// TIA Portal V18 export
VAR_GLOBAL   // PLC tag table "RemoteIO_DI_1"
   "iA-Loading-02Detection" AT %I1000.0 : Bool;   // A-转盘上料-02切料位检测
   "iA-Loading-02GripperTakeDetection" AT %I1000.1 : Bool;   // A-转盘上料-02夹爪取料位检测
   "iA-Loading-02PipeDetection" AT %I1000.2 : Bool;   // A-转盘上料-02料管检测
   "RESERVE_I1000.3" AT %I1000.3 : Bool;   // 备用_I1000.3
   "iA-Loading-02HorizontalCylinderInWP" AT %I1000.4 : Bool;   // A-转盘上料-02水平移栽气缸工作位
   "iA-Loading-02HorizontalCylinderInHP" AT %I1000.5 : Bool;   // A-转盘上料-02水平移栽气缸原始位
   "iA-Loading-02UpDownTakeCylinderInWP" AT %I1000.6 : Bool;   // A-转盘上料-02上下取料气缸工作位
   "iA-Loading-02UpDownTakeCylinderInHP" AT %I1000.7 : Bool;   // A-转盘上料-02上下取料气缸原始位
   "iB-PressFitting-02GripperCylinderInWP" AT %I1001.0 : Bool;   // B-压装模组-02夹爪气缸工作位
   "iB-PressFitting-02GripperCylinderInHP" AT %I1001.1 : Bool;   // B-压装模组-02夹爪气缸原始位
   "iB-PressFitting-02DownRingDetection" AT %I1001.2 : Bool;   // 备用_I1001.2
   "RESERVE_I1001.3" AT %I1001.3 : Bool;   // 备用_I1001.3
   "RESERVE_I1001.4" AT %I1001.4 : Bool;   // 备用_I1001.4
   "RESERVE_I1001.5" AT %I1001.5 : Bool;   // 备用_I1001.5
   "RESERVE_I1001.6" AT %I1001.6 : Bool;   // 备用_I1001.6
   "RESERVE_I1001.7" AT %I1001.7 : Bool;   // 备用_I1001.7
   "iB-PressFitting-02CylinderInWP" AT %I1002.0 : Bool;   // B-压装模组-02中转气缸工作位
   "iB-PressFitting-02CylinderInHP" AT %I1002.1 : Bool;   // B-压装模组-02中转气缸原始位
   "iB-PressFitting-02UpRingDetection" AT %I1002.2 : Bool;   // B-压装模组-02shaft有无检测
   "iB-PressFitting-02ShaftDetection" AT %I1002.3 : Bool;   // B-压装模组-02ring有无检测
   "RESERVE_I1002.4" AT %I1002.4 : Bool;   // 备用_I1002.4
   "RESERVE_I1002.5" AT %I1002.5 : Bool;   // 备用_I1002.5
   "RESERVE_I1002.6" AT %I1002.6 : Bool;   // 备用_I1002.6
   "RESERVE_I1002.7" AT %I1002.7 : Bool;   // 备用_I1002.7
   "iE-NG-02NGLocationCylinderInWP" AT %I1003.0 : Bool;   // E-NG料盒-02NG定位气缸工作位
   "iE-NG-02NGLocationCylinderInHP" AT %I1003.1 : Bool;   // E-NG料盒-02NG定位气缸原始位
   "iE-NG-03ShaftDispenseNGDetection" AT %I1003.2 : Bool;   // E-NG中转位-03shaft点胶NG有无检测
   "iE-NG-03MagnetDispenseNGDetection" AT %I1003.3 : Bool;   // E-NG中转位-03magnet点胶NG有无检测
   "iE-NG-02Detection" AT %I1003.4 : Bool;   // E-NG料盒-02到位检测
   "iC-GlueServoHomePos" AT %I1003.5 : Bool;   // 备用_I1003.5 / C-涂胶伺服原点
   "RESERVE_I1003.6" AT %I1003.6 : Bool;   // 备用_I1003.6
   "RESERVE_I1003.7" AT %I1003.7 : Bool;   // 备用_I1003.7
   "iC-LocationCylinderInWP" AT %I1004.0 : Bool;   // C-涂胶定位模组标准气缸工作位
   "iC-LocationCylinderInHP" AT %I1004.1 : Bool;   // C-涂胶定位模组标准气缸原始位
   "iC-LocationShaftDetection" AT %I1004.2 : Bool;   // C-涂胶定位模组shaft有无检测
   "iE-NG-01Detection" AT %I1004.3 : Bool;   // 备用_I1004.3 / E-NG料盒-01到位检测
   "iE-NG-01NGLocationCylinderInWP" AT %I1004.4 : Bool;   // E-NG料盒-01NG定位气缸工作位
   "iE-NG-01NGLocationCylinderInHP" AT %I1004.5 : Bool;   // E-NG料盒-01NG定位气缸原始位
   "RESERVE_I1004.6" AT %I1004.6 : Bool;   // E-NG料盒-01到位检测 / 备用_I1004.6
   "RESERVE_I1004.7" AT %I1004.7 : Bool;   // 备用_I1004.7
   "iB-PressFitting-01GripperCylinderInWP" AT %I1005.0 : Bool;   // B-压装模组-01夹爪气缸工作位
   "iB-PressFitting-01GripperCylinderInHP" AT %I1005.1 : Bool;   // B-压装模组-01夹爪气缸原始位
   "iB-PressFitting-01DownRingDetection" AT %I1005.2 : Bool;   // 备用_I1005.2
   "RESERVE_I1005.3" AT %I1005.3 : Bool;   // 备用_I1005.3
   "RESERVE_I1005.4" AT %I1005.4 : Bool;   // 备用_I1005.4
   "RESERVE_I1005.5" AT %I1005.5 : Bool;   // 备用_I1005.5
   "RESERVE_I1005.6" AT %I1005.6 : Bool;   // 备用_I1005.6
   "RESERVE_I1005.7" AT %I1005.7 : Bool;   // 备用_I1005.7
   "iB-PressFitting-01CylinderInWP" AT %I1006.0 : Bool;   // B-压装模组-01中转气缸工作位
   "iB-PressFitting-01CylinderInHP" AT %I1006.1 : Bool;   // B-压装模组-01中转气缸原始位
   "iB-PressFitting-01UpRingDetection" AT %I1006.2 : Bool;   // B-压装模组-01shaft有无检测-05
   "iB-PressFitting-01ShaftDetection" AT %I1006.3 : Bool;   // B-压装模组-01ring有无检测-06
   "iA-Rotating product Check" AT %I1006.4 : Bool;   // A-旋转处产品有无检测
   "RESERVE_I1006.5" AT %I1006.5 : Bool;   // 备用_I1006.5
   "RESERVE_I1006.6" AT %I1006.6 : Bool;   // 备用_I1006.6
   "RESERVE_I1006.7" AT %I1006.7 : Bool;   // 备用_I1006.7
   "iA-Loading-01Detection" AT %I1007.0 : Bool;   // A-转盘上料-01切料位检测
   "iA-Loading-01GripperTakeDetection" AT %I1007.1 : Bool;   // A-转盘上料-01夹爪取料位检测
   "iA-Loading-01PipeDetection" AT %I1007.2 : Bool;   // A-转盘上料-01料管检测
   "iA-Loading-01HorizontalCylinderInWP" AT %I1007.3 : Bool;   // A-转盘上料-01水平移栽气缸工作位
   "iA-Loading-01HorizontalCylinderInHP" AT %I1007.4 : Bool;   // A-转盘上料-01水平移栽气缸原始位
   "iA-Loading-01UpDownTakeCylinderInWP" AT %I1007.5 : Bool;   // A-转盘上料-01上下取料气缸工作位
   "iA-Loading-01UpDownTakeCylinderInHP" AT %I1007.6 : Bool;   // A-转盘上料-01上下取料气缸原始位
   "RESERVE_I1007.7" AT %I1007.7 : Bool;   // 备用_I1007.7
   "iE2-UnloadingPressNG_1" AT %I1008.0 : Bool;   // 备用_I1008.0
   "iE2-UnloadingPressNG_2" AT %I1008.1 : Bool;   // 备用_I1008.1
   "iE2-UnloadingPressNG_3" AT %I1008.2 : Bool;   // 备用_I1008.2
   "iE2-UnloadingPressNG_4" AT %I1008.3 : Bool;   // 备用_I1008.3
   "iE2-UnloadingPressNG_5" AT %I1008.4 : Bool;   // 备用_I1008.4
   "iE2-UnloadingMagentScanNG_1" AT %I1008.5 : Bool;   // 备用_I1008.5
   "iE2-UnloadingMagentScanNG_2" AT %I1008.6 : Bool;   // 备用_I1008.6
   "iE2-UnloadingMagentScanNG_3" AT %I1008.7 : Bool;   // 备用_I1008.7
   "iF-ROOBT3Gripper1CylinderInWP" AT %I1100.0 : Bool;   // F-ROBOT 3夹爪1夹爪气缸工作位
   "iF-ROOBT3Gripper1CylinderInHP" AT %I1100.1 : Bool;   // F-ROBOT 3夹爪1夹爪气缸原始位
   "iF-ROOBT3Gripper2CylinderInWP" AT %I1100.2 : Bool;   // F-ROBOT 3夹爪2夹爪气缸工作位
   "iF-ROOBT3Gripper2CylinderInHP" AT %I1100.3 : Bool;   // F-ROBOT 3夹爪2夹爪气缸原始位
   "RESERVE_I1100.4" AT %I1100.4 : Bool;   // 备用_I1100.4
   "RESERVE_I1100.5" AT %I1100.5 : Bool;   // 备用_I1100.5
   "RESERVE_I1100.6" AT %I1100.6 : Bool;   // 备用_I1100.6
   "RESERVE_I1100.7" AT %I1100.7 : Bool;   // 备用_I1100.7
   "iF-ROOBT3Gripper1Detection" AT %I1101.0 : Bool;   // F-ROBOT 3夹爪1料位检测
   "iF-ROOBT3Gripper2Detection-" AT %I1101.1 : Bool;   // F-ROBOT 3夹爪2料位检测-
   "RESERVE_I1101.2" AT %I1101.2 : Bool;   // 备用_I1101.2
   "RESERVE_I1101.3" AT %I1101.3 : Bool;   // 备用_I1101.3
   "RESERVE_I1101.4" AT %I1101.4 : Bool;   // 备用_I1101.4
   "RESERVE_I1101.5" AT %I1101.5 : Bool;   // 备用_I1101.5
   "RESERVE_I1101.6" AT %I1101.6 : Bool;   // 备用_I1101.6
   "RESERVE_I1101.7" AT %I1101.7 : Bool;   // 备用_I1101.7
   "iF-ROOBT2Gripper1CylinderInWP" AT %I1102.0 : Bool;   // F-ROBOT2夹爪1夹爪气缸工作位
   "iF-ROOBT2Gripper1CylinderInHP" AT %I1102.1 : Bool;   // F-ROBOT2夹爪1夹爪气缸原始位
   "iF-ROOBT2Gripper2CylinderInWP" AT %I1102.2 : Bool;   // F-ROBOT2夹爪2夹爪气缸工作位
   "iF-ROOBT2Gripper2CylinderInHP" AT %I1102.3 : Bool;   // F-ROBOT2夹爪2夹爪气缸原始位
   "RESERVE_I1102.4" AT %I1102.4 : Bool;   // 备用_I1102.4
   "RESERVE_I1102.5" AT %I1102.5 : Bool;   // 备用_I1102.5
   "RESERVE_I1102.6" AT %I1102.6 : Bool;   // 备用_I1102.6
   "RESERVE_I1102.7" AT %I1102.7 : Bool;   // 备用_I1102.7
   "iF-ROOBT2Gripper1Detection" AT %I1103.0 : Bool;   // F-ROBOT2夹爪1料位检测
   "iF-ROOBT2Gripper2Detection" AT %I1103.1 : Bool;   // F-ROBOT2夹爪2料位检测
   "RESERVE_I1103.2" AT %I1103.2 : Bool;   // 备用_I1103.2
   "RESERVE_I1103.3" AT %I1103.3 : Bool;   // 备用_I1103.3
   "RESERVE_I1103.4" AT %I1103.4 : Bool;   // 备用_I1103.4
   "RESERVE_I1103.5" AT %I1103.5 : Bool;   // 备用_I1103.5
   "RESERVE_I1103.6" AT %I1103.6 : Bool;   // 备用_I1103.6
   "RESERVE_I1103.7" AT %I1103.7 : Bool;   // 备用_I1103.7
   "iF-ROOBT1Gripper1CylinderInWP" AT %I1104.0 : Bool;   // F-ROBOT 1夹爪1夹爪气缸工作位
   "iF-ROOBT1Gripper1CylinderInHP" AT %I1104.1 : Bool;   // F-ROBOT 1夹爪1夹爪气缸原始位
   "iF-ROOBT1Gripper2CylinderInWP" AT %I1104.2 : Bool;   // F-ROBOT 1夹爪2夹爪气缸工作位
   "iF-ROOBT1Gripper2CylinderInHP" AT %I1104.3 : Bool;   // F-ROBOT 1夹爪2夹爪气缸原始位
   "RESERVE_I1104.4" AT %I1104.4 : Bool;   // 备用_I1104.4
   "RESERVE_I1104.5" AT %I1104.5 : Bool;   // 备用_I1104.5
   "RESERVE_I1104.6" AT %I1104.6 : Bool;   // 备用_I1104.6
   "RESERVE_I1104.7" AT %I1104.7 : Bool;   // 备用_I1104.7
   "iF-ROOBT1Gripper1Detection" AT %I1105.0 : Bool;   // F-ROBOT 1夹爪1料位检测
   "iF-ROOBT1Gripper2Detection" AT %I1105.1 : Bool;   // F-ROBOT 1夹爪2料位检测
   "iF-ROOBT1ShaftDetection" AT %I1105.2 : Bool;   // F-ROBOT 1shaft有无检测
   "RESERVE_I1105.3" AT %I1105.3 : Bool;   // 备用_I1105.3
   "RESERVE_I1105.4" AT %I1105.4 : Bool;   // 备用_I1105.4
   "RESERVE_I1105.5" AT %I1105.5 : Bool;   // 备用_I1105.5
   "RESERVE_I1105.6" AT %I1105.6 : Bool;   // 备用_I1105.6
   "RESERVE_I1105.7" AT %I1105.7 : Bool;   // 备用_I1105.7
   "iE2-UnloadingMagentScanNG_4" AT %I1009.0 : Bool;
   "iE2-UnloadingMagentScanNG_5" AT %I1009.1 : Bool;
   "iE2-UnloadingRingScanNG_1" AT %I1009.2 : Bool;
   "iE2-UnloadingRingScanNG_2" AT %I1009.3 : Bool;
   "iE2-UnloadingRingScanNG_3" AT %I1009.4 : Bool;
   "iE2-UnloadingRingScanNG_4" AT %I1009.5 : Bool;
   "iE2-UnloadingRingScanNG_5" AT %I1009.6 : Bool;
   "RESERVE_I1009.7" AT %I1009.7 : Bool;
   "iE1-UnloadingShaftPressNG_1" AT %I1010.0 : Bool;
   "iE1-UnloadingShaftPressNG_2" AT %I1010.1 : Bool;
   "iE1-UnloadingShaftPressNG_3" AT %I1010.2 : Bool;
   "iE1-UnloadingShaftPressNG_4" AT %I1010.3 : Bool;
   "iE1-UnloadingShaftPressNG_5" AT %I1010.4 : Bool;
   "iE1-UnloadingShaftScanNG_1" AT %I1010.5 : Bool;
   "iE1-UnloadingShaftScanNG_2" AT %I1010.6 : Bool;
   "iE1-UnloadingShaftScanNG_3" AT %I1010.7 : Bool;
   "iE1-UnloadingShaftScanNG_4" AT %I1011.0 : Bool;
   "iE1-UnloadingShaftScanNG_5" AT %I1011.1 : Bool;
   "iE1-UnloadingRingScanNG_1" AT %I1011.2 : Bool;
   "iE1-UnloadingRingScanNG_2" AT %I1011.3 : Bool;
   "iE1-UnloadingRingScanNG_3" AT %I1011.4 : Bool;
   "iE1-UnloadingRingScanNG_4" AT %I1011.5 : Bool;
   "iE1-UnloadingRingScanNG_5" AT %I1011.6 : Bool;
   "RESERVE_I1011.7" AT %I1011.7 : Bool;
END_VAR
